Fanuc KAREL source: kx00014.KL

-- PROVISIONAL review KL for V940-1; original PC SHA256 df81555cd101cb989d71a9d3a2e61b9f3c6a6dd7eb052f8139699cd6d9c9bafe
-- Incomplete behavior may be omitted. Consult companion uncertainty JSON. Do not deploy.
PROGRAM KX00014
%NOLOCKGROUP
VAR
  I : INTEGER
  J : INTEGER
  B : BOOLEAN
  F : FILE
  S : STRING[80]
-- UNRESOLVED_DECL P type=000102
BEGIN
  -- V9_ZERO_TABLE_METADATA_HINT layout=0001; no indexed target words; source/name/runtime held
  -- UNRESOLVED_PC offsets 5-7; opcodes 9D,3C
  -- UNRESOLVED_PC offsets 12-16; opcodes 7F
END KX00014
